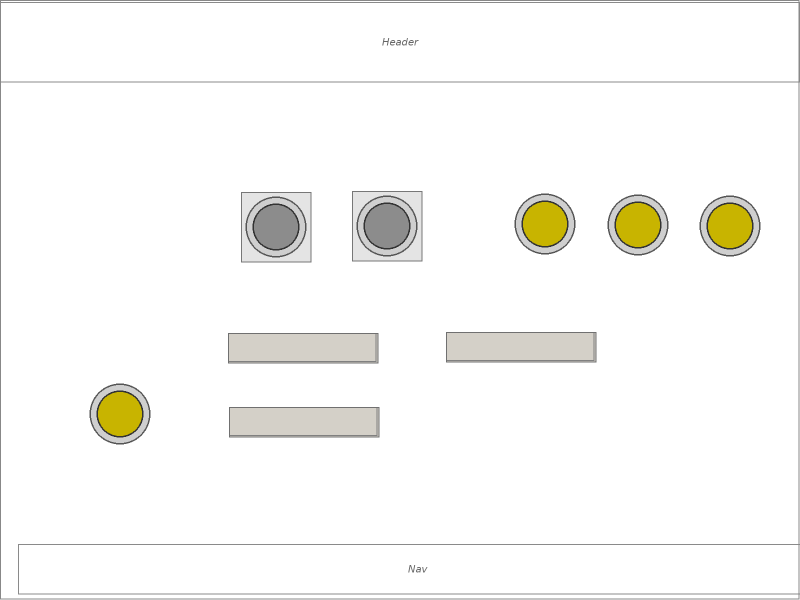
VISUALIZATION Visualization  // 800x600
    PushSwitch (241,192 70x70), variable: Variables.start, behaviour: TOGGLE, style: Switch-PushSwitch-Gray
    PushSwitch (352,191 70x70), variable: Variables.stop, behaviour: TOGGLE, style: Switch-PushSwitch-Gray
    Lamp1 (603,190 70x70), variable: Variables.motor2, style: Lamp-Lamp1-Yellow
    Lamp1 (510,189 70x70), variable: Variables.motor1, style: Lamp-Lamp1-Yellow
    Button (228,333 150x30)
        OnMouseDown: toggle Variables.start
        OnMouseUp: toggle Variables.start
    Lamp1 (695,191 70x70), variable: Variables.motor3, style: Lamp-Lamp1-Yellow
    Button (446,332 150x30)
        OnMouseDown: toggle Variables.stop
        OnMouseUp: toggle Variables.stop
    Lamp1 (85,379 70x70), variable: Variables.LED, style: Lamp-Lamp1-Yellow
    Button (229,407 150x30)
        OnMouseDown: toggle Variables.Button
        OnMouseUp: toggle Variables.Button
    Frame (0,2 800x80)
        shows Header()
    Frame (18,544 800x50)
        shows Nav()
END_VISUALIZATION

(* stored: Version 1.1.0.1, ProductVersion 3.1.4024.12
   Visu Visualization: Id {c387dfae-170e-4ace-9d72-17867440cb50} *)
